FUNCTION_BLOCK SWITCHER (* Basic Function Block Type *)
  (* Standard: 61499-2 *)
  (* Version 0.3, 2009-09-15, JHC, Holobloc Inc, Changed transition priorities. *)
  (* Version 0.2, 2003-12-04, JHC, Rockwell Automation, Renamed for better indexing. *)
  (* Version 0.1, 2002-11-05, JHC, Rockwell Automation, Corrected missing ST element in Algorithm REQ. *)
  (* Version 0.0, 2000-05-30, JHC, Rockwell Automation *)
  (* Compiler header: package fb.rt.icaru; *)
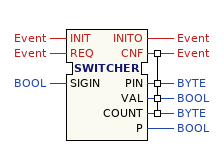
  EVENT_INPUT
    INIT; (* Initialization Request *)
    REQ; (* Normal Execution Request *)
  END_EVENT
  EVENT_OUTPUT
    INITO; (* Initialization Confirm *)
    CNF WITH PIN, VAL, COUNT; (* Execution Confirmation *)
  END_EVENT
  VAR_INPUT
    SIGIN : BOOL;
  END_VAR
  VAR_OUTPUT
    PIN : BYTE;
    VAL : BOOL;
    COUNT : BYTE;
    P : BOOL;
  END_VAR
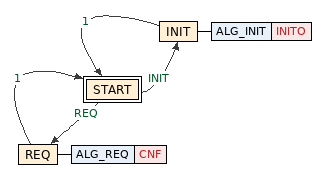
  EC_STATES
    START; (* Initial State *)
    INIT : ALG_INIT -> INITO; (* Initialization *)
    REQ : ALG_REQ -> CNF; (* Normal execution *)
  END_STATES
  EC_TRANSITIONS
    INIT TO START := 1;
    START TO REQ := REQ;
    START TO INIT := INIT;
    REQ TO START := 1;
  END_TRANSITIONS
  ALGORITHM ALG_INIT IN ST: (* Initialization algorithm *)
COUNT:=0;
VAL:=1;
  END_ALGORITHM
  ALGORITHM ALG_REQ IN ST: (* Normally executed algorithm *)
IF NOT SIGIN AND P THEN
 P := 0;
 COUNT := COUNT + 1;
 IF (COUNT > 3) THEN
   COUNT := 0;
   VAL := NOT VAL;
 END_IF;
 PIN := 200 + COUNT;
END_IF;
IF SIGIN THEN
 P := 1;
END_IF;
  END_ALGORITHM
END_FUNCTION_BLOCK
